FUNCTION GenerateOscillation : REAL
VAR_INPUT
	rRand: REAL;
END_VAR
VAR
END_VAR

rRand := (RAND() - 0.5) * rOscillationRange * 2; // Generates random value between -rOscillationRange and +rOscillationRange
    GenerateOscillation := rRand;

END_FUNCTION

(* stored: Version 1.1.0.1, ProductVersion 3.1.4024.13
   POU GenerateOscillation: Id {534cb044-12f8-42ed-91e6-9701a1a88487}, SpecialFunc None *)
